FUNCTION_BLOCK Sensor
VAR_INPUT
END_VAR
VAR_OUTPUT
	bSignal  : BOOL;
END_VAR
VAR
	fbSignal : BoolIn;
END_VAR

bSignal := fbSignal.getValue;

PROPERTY getSignal : I_StepCondition
GET
getSignal := fbSignal;
END_GET
END_PROPERTY

END_FUNCTION_BLOCK

(* stored: Version 1.1.0.1, ProductVersion 3.1.4024.2
   POU Sensor: Id {ecf36537-b594-4d9d-9568-9f92fc6eecfa}, SpecialFunc None
   Property getSignal: Id {d2f422ba-76f1-4996-bc13-0bbe2b33b8cb}
   Get Get: Id {a22c8bbd-ba75-4175-8f2e-afc0bcf15c4d} *)
